(* IEC 61131-3 sources: LASAL/Class/Encoders, 1 file *)

(* ---- Encoders.st ---- *)
(*!
<Class
	Name               = "Encoders"
	Revision           = "0.0"
	RealtimeTask       = "true"
	DefRealtime        = "1 ms"
	CyclicTask         = "false"
	BackgroundTask     = "false"
	Sigmatek           = "false"
	OSInterface        = "false"
	HighPriority       = "false"
	Automatic          = "false"
	UpdateMode         = "Prescan"
	SharedCommandTable = "true"
	Objectsize         = "(480,300)">
	<Channels>
		<Server Name="DIV" Visualized="false" Initialize="true" WriteProtected="false" Retentive="File"/>
		<Server Name="InvertOutput" Visualized="false" Initialize="true" WriteProtected="false" Retentive="File"/>
		<Server Name="KV" Visualized="false" Initialize="true" WriteProtected="false" Retentive="File"/>
		<Server Name="MUL" Visualized="false" Initialize="true" WriteProtected="false" Retentive="File"/>
		<Server Name="Target" Visualized="false" Initialize="false" WriteProtected="false" Retentive="false"/>
		<Client Name="pos_in_fixed" Required="true" Internal="false"/>
		<Client Name="pos_in_steppermotor" Required="true" Internal="false"/>
		<Client Name="Pos_out" Required="true" Internal="false"/>
		<Client Name="Speed_out" Required="true" Internal="false"/>
	</Channels>
</Class>
*)
Encoders : CLASS
  //Servers:
	Target 	: SvrChCmd_DINT;
	KV 	: SvrCh_DINT;
	MUL 	: SvrCh_DINT;
	DIV 	: SvrCh_DINT;
	InvertOutput 	: SvrCh_DINT;
  //Clients:
	pos_in_fixed 	: CltCh_DINT;
	pos_in_steppermotor 	: CltCh_DINT;
	Speed_out 	: CltCh_DINT;
	Pos_out 	: CltCh_DINT;
  //Variables:
		Stepper_to_encoder 	: DINT;
		Delta 	: DINT;
		OldPos 	: DINT;
		NewPos 	: DINT;
  //Functions:

	FUNCTION VIRTUAL GLOBAL Init;

	FUNCTION VIRTUAL GLOBAL RtWork
		VAR_INPUT
			EAX 	: UDINT;
		END_VAR
		VAR_OUTPUT
			state (EAX) 	: UDINT;
		END_VAR;
  //Tables:
	FUNCTION @STD
		VAR_OUTPUT
			ret_code	: CONFSTATES;
		END_VAR;
	FUNCTION GLOBAL TAB @CT_;
END_CLASS;

FUNCTION VIRTUAL GLOBAL Encoders::Init
if div=0 then div:=1000;end_if;
END_FUNCTION

FUNCTION VIRTUAL GLOBAL Encoders::RtWork
	VAR_INPUT
		EAX 	: UDINT;
	END_VAR
	VAR_OUTPUT
		state (EAX) 	: UDINT;
	END_VAR
  pos_in_fixed:=pos_in_fixed.Read();
  Pos_out:=Pos_out.Read();

  pos_in_steppermotor:=pos_in_steppermotor.Read();
  Stepper_to_encoder:=pos_in_steppermotor*mul/div;

  NewPos:=pos_in_fixed-Stepper_to_encoder;
  Delta:=NewPos-OldPos;
  OldPos:=NewPos;

  Target+=Delta*InvertOutput;

  Speed_out:=(Target-Pos_out)*kv;

  Speed_out.Write(input:=Speed_out);

	state := READY;

END_FUNCTION
